(* IEC 61131-3 sources: ElnaAutomator/ExampleProject/Functions, 19 files *)

(* ---- AnyAnalogsNs.st ---- *)
FUNCTION AnyAnalogsNs : BOOL

VAR_INPUT
	Ai : AiConfig;
END_VAR

VAR
	statusAi : TYPE_StatusAi;
END_VAR

AnyAnalogsNs :=
((Ai.A1.interval < statusAi.Normal) AND NOT Ai.A1.Remont) OR
((Ai.A2.interval < statusAi.Normal) AND NOT Ai.A2.Remont);

(* ---- AnyAnalogsPs.st ---- *)
FUNCTION AnyAnalogsPs : BOOL

VAR_INPUT
	Ai : AiConfig;
END_VAR

VAR
	statusAi : TYPE_StatusAi;
END_VAR

AnyAnalogsPs :=
Ai.A1.interval = statusAi.HW OR
Ai.A2.interval = statusAi.HW OR
Ai.A1.interval = statusAi.LW OR
Ai.A2.interval = statusAi.LW;

(* ---- AnyDiscretNs.st ---- *)
FUNCTION AnyDiscretNs : BOOL

VAR_INPUT
	Di : DiConfig;
END_VAR

AnyDiscretNs :=
((Di.Di.reliability <> 255) OR
(Di.Di1.reliability <> 255) OR
(Di.Di2.reliability <> 255) OR
(Di.Di3.reliability <> 255) OR
(Di.Di4.reliability <> 255));

(* ---- AnyDiscretPs.st ---- *)
FUNCTION AnyDiscretPs : BOOL

VAR_INPUT
	Im : ImConfig;
END_VAR

AnyDiscretPs :=
Im.SingleSignals.SI0.Q;

(* ---- AnyProtectionInRemont.st ---- *)
FUNCTION AnyProtectionInRemont : BOOL

VAR_INPUT
	Protections : ProtectionsConfig;
END_VAR

AnyProtectionInRemont :=
Protections.Ap1.Remont OR
Protections.AiP1.Remont OR
Protections.AiP2.Remont OR
Protections.AiP3.Remont OR
Protections.DiP1.Remont OR
Protections.DiP2.Remont OR
Protections.DiP3.Remont OR
Protections.DiP4.Remont OR
Protections.DiP5.Remont;

(* ---- AnyProtectionSignaling.st ---- *)
FUNCTION AnyProtectionSignaling : BOOL

VAR_INPUT
	Protections : ProtectionsConfig;
END_VAR

AnyProtectionSignaling :=
Protections.Ap1.Signaling OR
Protections.AiP1.Signaling OR
Protections.AiP2.Signaling OR
Protections.AiP3.Signaling OR
Protections.DiP1.Signaling OR
Protections.DiP2.Signaling OR
Protections.DiP3.Signaling OR
Protections.DiP4.Signaling OR
Protections.DiP5.Signaling;

(* ---- AutoRunProtections.st ---- *)
FUNCTION AutoRunProtections : BOOL

VAR_IN_OUT
	Protections : ProtectionsConfig;
END_VAR

RunAiProtection(Protections.Ap1);
RunAiProtection(Protections.AiP2);
RunDiProtection(Protections.DiP1);
RunDiProtection(Protections.DiP2);
RunDiProtection(Protections.DiP3);

(* ---- BlockAllIm.st ---- *)
FUNCTION BlockAllIm : BOOL

VAR_IN_OUT
	IM : ImConfig;
END_VAR

IF NOT IM.Kran1.inOpcCommandsDisabled THEN IM.Kran1.inOpcCommandsDisabled := TRUE; END_IF;
IF NOT IM.Kran4.inOpcCommandsDisabled THEN IM.Kran4.inOpcCommandsDisabled := TRUE; END_IF;
IF NOT IM.Kran2.inOpcCommandsDisabled THEN IM.Kran2.inOpcCommandsDisabled := TRUE; END_IF;
IF NOT IM.Kran3.inOpcCommandsDisabled THEN IM.Kran3.inOpcCommandsDisabled := TRUE; END_IF;
IF NOT IM.Nu.inOpcCommandsDisabled THEN IM.Nu.inOpcCommandsDisabled := TRUE; END_IF;
IF NOT IM.Nu2.inOpcCommandsDisabled THEN IM.Nu2.inOpcCommandsDisabled := TRUE; END_IF;
IF NOT IM.Avom1.inOpcCommandsDisabled THEN IM.Avom1.inOpcCommandsDisabled := TRUE; END_IF;
IF NOT IM.Avom2.inOpcCommandsDisabled THEN IM.Avom2.inOpcCommandsDisabled := TRUE; END_IF;
IF NOT IM.Avom3.inOpcCommandsDisabled THEN IM.Avom3.inOpcCommandsDisabled := TRUE; END_IF;
IF NOT IM.Avom4.inOpcCommandsDisabled THEN IM.Avom4.inOpcCommandsDisabled := TRUE; END_IF;
IF NOT IM.Mv.inOpcCommandsDisabled THEN IM.Mv.inOpcCommandsDisabled := TRUE; END_IF;
IF NOT IM.SectionSwitch1.inOpcCommandsDisabled THEN IM.SectionSwitch1.inOpcCommandsDisabled := TRUE; END_IF;

(* ---- BlockAllProtections.st ---- *)
FUNCTION BlockAllProtections : BOOL

VAR_IN_OUT
	Protections : ProtectionsConfig;
END_VAR

Protections.Ap1.inOpcCommandsDisabled := TRUE;
Protections.AiP1.inOpcCommandsDisabled := TRUE;
Protections.AiP2.inOpcCommandsDisabled := TRUE;
Protections.AiP3.inOpcCommandsDisabled := TRUE;
Protections.DiP1.inOpcCommandsDisabled := TRUE;
Protections.DiP2.inOpcCommandsDisabled := TRUE;
Protections.DiP3.inOpcCommandsDisabled := TRUE;
Protections.DiP4.inOpcCommandsDisabled := TRUE;
Protections.DiP5.inOpcCommandsDisabled := TRUE;

(* ---- DisableAiLimits.st ---- *)
FUNCTION DisableAiLimits : BOOL

VAR_IN_OUT
	Ai : AiConfig;
END_VAR

Ai.A1.Disabled_LA := TRUE;
Ai.A2.Disabled_LA := TRUE;
Ai.A1.Disabled_LW := TRUE;
Ai.A2.Disabled_LW := TRUE;

(* ---- DIwValue_Diag.st ---- *)
FUNCTION DIwValue_Diag : UDINT

VAR_INPUT
	val1 : UINT;
	val2 : UINT;
END_VAR

VAR
	val1_tmp : DWORD;
	val2_tmp : DWORD;
END_VAR

(* Переставлем биты value и reability местами для корректного отображения в MasterScada *)

val1_tmp:=(SHL(UINT_TO_DWORD(val1),1) AND 16#AAAA) OR (SHR(UINT_TO_DWORD(val1),1) AND 16#5555);

val2_tmp:=(SHL(UINT_TO_DWORD(val2),1) AND 16#AAAA) OR (SHR(UINT_TO_DWORD(val2),1) AND 16#5555);

(* Вместо reability = 1 посдставляем инверсию сигнала в виде , если нет reability тогда обрыв = 1 для MasterScada *)

DIwValue_Diag:= DWORD_TO_UDINT((val1_tmp OR shl(val2_tmp, 16)) XOR 16#55555555);

(* ---- EnableAiLimits.st ---- *)
FUNCTION EnableAiLimits : BOOL

VAR_IN_OUT
	Ai : AiConfig;
END_VAR

Ai.A1.Disabled_LA := FALSE;
Ai.A2.Disabled_LA := FALSE;
Ai.A1.Disabled_LW := FALSE;
Ai.A2.Disabled_LW := FALSE;

(* ---- NsCepeiControl.st ---- *)
FUNCTION NsCepeiControl : BOOL

VAR_INPUT
	IM : ImConfig;
END_VAR

NsCepeiControl := NOT (
	IM.Kran1.reliability OR
	IM.Kran4.reliability OR
	IM.Kran2.reliability OR
	IM.Kran3.reliability OR
	IM.Nu.reliability OR
	IM.Nu2.reliability OR
	IM.Avom1.reliability OR
	IM.Avom2.reliability OR
	IM.Avom3.reliability OR
	IM.Avom4.reliability OR
	IM.Mv.reliability OR
	IM.SectionSwitch1.reliability);

(* ---- NsCepeiUpravlenya.st ---- *)
FUNCTION NsCepeiUpravlenya : BOOL

VAR_INPUT
	IM : ImConfig;
END_VAR

NsCepeiUpravlenya := (
	IM.Kran4.Sz OR
	IM.Kran2.Sz OR
	IM.Kran3.So OR
	IM.Nu.breakCmdOn OR
	IM.Nu2.breakCmdOn OR
	IM.Avom1.breakCmdOn OR
	IM.Avom2.breakCmdOn OR
	IM.Avom3.breakCmdOn OR
	IM.Avom4.breakCmdOn OR
	IM.Mv.breakCmdOn);

(* ---- RemontAllProtections.st ---- *)
FUNCTION RemontAllProtections : BOOL

VAR_IN_OUT
	Protections : ProtectionsConfig;
END_VAR

VAR CONSTANT
	cmdRemont : WORD := 4;
END_VAR

Protections.Ap1.inCommand_Alg := cmdRemont;
Protections.AiP1.inCommand_Alg := cmdRemont;
Protections.AiP2.inCommand_Alg := cmdRemont;
Protections.AiP3.inCommand_Alg := cmdRemont;
Protections.DiP1.inCommand_Alg := cmdRemont;
Protections.DiP2.inCommand_Alg := cmdRemont;
Protections.DiP3.inCommand_Alg := cmdRemont;
Protections.DiP4.inCommand_Alg := cmdRemont;
Protections.DiP5.inCommand_Alg := cmdRemont;

(* ---- ResetAllProtections.st ---- *)
FUNCTION ResetAllProtections : BOOL

VAR_IN_OUT
	Protections : ProtectionsConfig;
END_VAR

ResetAiProtection(Protections.Ap1);
ResetAiProtection(Protections.AiP1);
ResetAiProtection(Protections.AiP2);
ResetAiProtection(Protections.AiP3);
ResetDiProtection(Protections.DiP1);
ResetDiProtection(Protections.DiP2);
ResetDiProtection(Protections.DiP3);
ResetDiProtection(Protections.DiP4);
ResetDiProtection(Protections.DiP5);

(* ---- ResetAllSignaling.st ---- *)
FUNCTION ResetAllSignaling : BOOL

VAR_IN_OUT
	Protections : ProtectionsConfig;
END_VAR

IF Protections.Ap1.Signaling THEN
	ResetAiProtection(Protections.Ap1); END_IF;
IF Protections.AiP1.Signaling THEN
	ResetAiProtection(Protections.AiP1); END_IF;
IF Protections.AiP2.Signaling THEN
	ResetAiProtection(Protections.AiP2); END_IF;
IF Protections.AiP3.Signaling THEN
	ResetAiProtection(Protections.AiP3); END_IF;
IF Protections.DiP1.Signaling THEN
	ResetDiProtection(Protections.DiP1); END_IF;
IF Protections.DiP2.Signaling THEN
	ResetDiProtection(Protections.DiP2); END_IF;
IF Protections.DiP3.Signaling THEN
	ResetDiProtection(Protections.DiP3); END_IF;
IF Protections.DiP4.Signaling THEN
	ResetDiProtection(Protections.DiP4); END_IF;
IF Protections.DiP5.Signaling THEN
	ResetDiProtection(Protections.DiP5); END_IF;

(* ---- UnBlockAllIm.st ---- *)
FUNCTION UnBlockAllIm : BOOL

VAR_IN_OUT
	IM : ImConfig;
END_VAR

IF IM.Kran1.inOpcCommandsDisabled THEN IM.Kran1.inOpcCommandsDisabled := FALSE; END_IF;
IF IM.Kran4.inOpcCommandsDisabled THEN IM.Kran4.inOpcCommandsDisabled := FALSE; END_IF;
IF IM.Kran2.inOpcCommandsDisabled THEN IM.Kran2.inOpcCommandsDisabled := FALSE; END_IF;
IF IM.Kran3.inOpcCommandsDisabled THEN IM.Kran3.inOpcCommandsDisabled := FALSE; END_IF;
IF IM.Nu.inOpcCommandsDisabled THEN IM.Nu.inOpcCommandsDisabled := FALSE; END_IF;
IF IM.Nu2.inOpcCommandsDisabled THEN IM.Nu2.inOpcCommandsDisabled := FALSE; END_IF;
IF IM.Avom1.inOpcCommandsDisabled THEN IM.Avom1.inOpcCommandsDisabled := FALSE; END_IF;
IF IM.Avom2.inOpcCommandsDisabled THEN IM.Avom2.inOpcCommandsDisabled := FALSE; END_IF;
IF IM.Avom3.inOpcCommandsDisabled THEN IM.Avom3.inOpcCommandsDisabled := FALSE; END_IF;
IF IM.Avom4.inOpcCommandsDisabled THEN IM.Avom4.inOpcCommandsDisabled := FALSE; END_IF;
IF IM.Mv.inOpcCommandsDisabled THEN IM.Mv.inOpcCommandsDisabled := FALSE; END_IF;
IF IM.SectionSwitch1.inOpcCommandsDisabled THEN IM.SectionSwitch1.inOpcCommandsDisabled := FALSE; END_IF;

(* ---- UnBlockAllProtections.st ---- *)
FUNCTION UnBlockAllProtections : BOOL

VAR_IN_OUT
	Protections : ProtectionsConfig;
END_VAR

protections.Ap1.inOpcCommandsDisabled := FALSE;
protections.AiP1.inOpcCommandsDisabled := FALSE;
protections.AiP2.inOpcCommandsDisabled := FALSE;
protections.AiP3.inOpcCommandsDisabled := FALSE;
protections.DiP1.inOpcCommandsDisabled := FALSE;
protections.DiP2.inOpcCommandsDisabled := FALSE;
protections.DiP3.inOpcCommandsDisabled := FALSE;
protections.DiP4.inOpcCommandsDisabled := FALSE;
protections.DiP5.inOpcCommandsDisabled := FALSE;
